//==================================================================================================
//								RJM Maszyny sp. z o.o.
//									13.05.2022
//
//	Obsługa czujnika
//	v1.0	|| TC v 3.1.4024.22		|| - pierwsza wersja
//==================================================================================================
INTERFACE I_Czujnik

//==================================================================================================
//								RJM Maszyny sp. z o.o.
//									13.05.2022
//
//	Sprawdzenie czy aktywny
//	v1.0	|| TC v 3.1.4024.22		|| - pierwsza wersja
//==================================================================================================
PROPERTY CzyAktywny : BOOL
GET
END_GET
END_PROPERTY

END_INTERFACE

(* stored: Version 1.1.0.1, ProductVersion 3.1.4024.11
   Itf I_Czujnik: Id {3424d7ca-b997-4079-8e5a-d210800efc9f}
   Property CzyAktywny: Id {0f6431ef-e80b-4ffb-9a56-cab398117bf1}
   Get Get: Id {6c3af1c3-6152-4478-b468-1bd69fe7e424} *)
